{region '#Template'}
	{attribute 'Version' := '1.2.1.0'}
	{attribute 'Tags' := '"LCID": "1031", "Text": "General, Cabinet, Control cabinet, Acknowledgement"'}
	{attribute 'Tags' := '"LCID": "1033", "Text": "General, Cabinet, Control cabinet, Acknowledgement"'}
	{attribute 'Using' := '"Type": "Template", "URI": "EC_AMEV"'}
	{attribute 'Description' := '"LCID": "1031", "Text": "Schaltschrank Quittierung"'}
	{attribute 'Description' := '"LCID": "1033", "Text": "Control cabinet acknowledgement"'}
{endregion}
FUNCTION_BLOCK FB_BA_ControlCabinetBasic EXTENDS FB_BA_View
VAR
	// By default, the entire project structure can be acknowledged.
	// There may be constellations (e.g. multiple control cabinets) where only one part of the project structure (e.g. multiple buildings) has to be acknowledged.
	// > In this case separete parts can be assigned here: 
	iAckView1				: I_BA_View;
	iAckView2				: I_BA_View;
	iAckView3				: I_BA_View;
END_VAR
VAR_INPUT CONSTANT
	LampFault				: FB_BA_ActuatorCmd;		
	AckButton				: FB_BA_CombinationBI_BV;													
	RstHw					: FB_BA_ActuatorCmd;														
END_VAR
VAR				
	bIsDisturbed			: BOOL;
	bHasUnackEvent			: BOOL;
	bBlink					: BOOL;
	tAlmLampImpuls			: FB_BA_Blink;						
	tpResetHw				: TP;	
	rtrigRstSwi				: R_TRIG;
	bTrigRstSwi				: BOOL;
	rtrigRstButton			: R_TRIG;
	bTrigRstButton			: BOOL;	
END_VAR

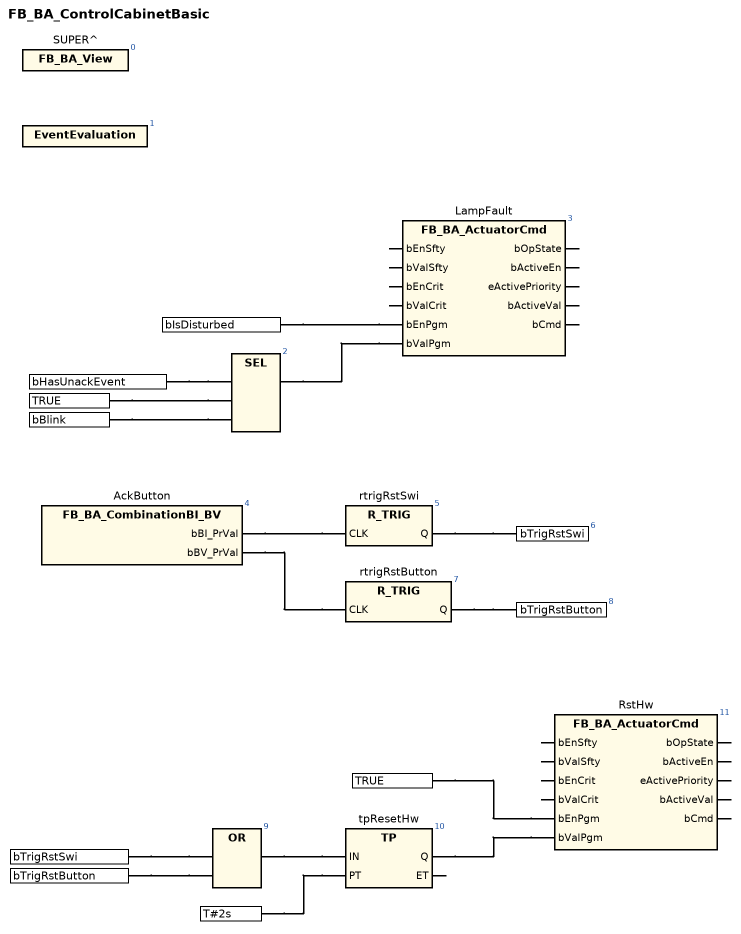
SUPER^(); // FB_BA_View
EventEvaluation();
LampFault(bEnPgm := bIsDisturbed, bValPgm := SEL(bHasUnackEvent, TRUE, bBlink)); // FB_BA_ActuatorCmd
AckButton(); // FB_BA_CombinationBI_BV
rtrigRstSwi(CLK := AckButton.bBI_PrVal); // R_TRIG
bTrigRstSwi := rtrigRstSwi.Q;
rtrigRstButton(CLK := AckButton.bBV_PrVal); // R_TRIG
bTrigRstButton := rtrigRstButton.Q;
tpResetHw(IN := bTrigRstSwi OR bTrigRstButton, PT := T#2s); // TP
RstHw(bEnPgm := TRUE, bValPgm := tpResetHw.Q); // FB_BA_ActuatorCmd

METHOD PRIVATE Ack
VAR_INPUT
	iView			: I_BA_View;
END_VAR
IF (iView <> 0) THEN
	iView.AcknowledgeObjectsPLC := (bTrigRstSwi) OR (bTrigRstButton);	
END_IF
END_METHOD

METHOD PRIVATE EventEvaluation
VAR
	_iView			: I_BA_View;
END_VAR
bIsDisturbed := FALSE;
bHasUnackEvent := FALSE;

IF (iAckView1 = 0) AND (iAckView2 = 0) AND (iAckView3 = 0) THEN
	// Treat project structure via root-object:
	Ack(BA_Globals.Top);
	GetErrors(BA_Globals.Top);
ELSE
	// Treat each defined object:
	Ack(iAckView1);
	GetErrors(iAckView1);
	
	Ack(iAckView2);
	GetErrors(iAckView2);
	
	Ack(iAckView3);
	GetErrors(iAckView3);
END_IF

// Generate alarm lamp impulse:
tAlmLampImpuls();

bBlink := tAlmLampImpuls.bQ;
END_METHOD

METHOD FB_init : BOOL
VAR_INPUT
	bInitRetains : BOOL; // if TRUE, the retain variables are initialized (warm start / cold start)
	bInCopyCode : BOOL;  // if TRUE, the instance afterwards gets moved into the copy code (online change)
END_VAR
LampFault.iParent							:= THIS^;
LampFault.iLabel							:= LblCmpGeneral.ControlCabinet_LampFault;			
LampFault.sObjectName						:= '{Idx=01}';
LampFault.eDPADMode							:= E_BA_DPADMode.eInclude;																						
LampFault.Cmd.iLabel						:= LblCmpGeneral.ControlCabinet_LampFault_Cmd;			
LampFault.Cmd.sObjectName					:= '{Idx=01}';	
LampFault.Cmd.ePolarity						:= E_BA_Polarity.eNormal;
LampFault.Cmd.eFeedbackPolarity				:= E_BA_Polarity.eNormal;
LampFault.Cmd.eOverriddenPolarity			:= E_BA_Polarity.eReverse;
LampFault.Cmd.sActiveText 					:= txtEvent_On;
LampFault.Cmd.sInactiveText 				:= txtEvent_Off;
LampFault.Cmd.nEventClassID					:= EC_ID.NC40;
LampFault.Cmd.aEventTransitionText[1]		:= txtEvent_Disturb;
LampFault.Cmd.aEventTransitionText[2]		:= txtEvent_None;
LampFault.Cmd.aEventTransitionText[3]		:= txtEvent_Normal;
LampFault.Cmd.bEventDetectionEnable			:= FALSE;
LampFault.Cmd.eEnPlantLock					:= E_BA_LockPriority.eNoLock;	

AckButton.iParent							:= THIS^;		
AckButton.iLabel 							:= LblCmpGeneral.ControlCabinet_AckButton;	
AckButton.sObjectName						:= '{Idx=01}';
AckButton.eDPADMode							:= E_BA_DPADMode.eInclude;																						
AckButton.Input.iLabel						:= LblCmpGeneral.ControlCabinet_AckButton_Input;
AckButton.Input.ePolarity					:= E_BA_Polarity.eNormal;
AckButton.Input.bEventDetectionEnable		:= FALSE;
AckButton.Value.iLabel						:= LblCmpGeneral.ControlCabinet_AckButton_Value;
AckButton.Value.eToggleMode 				:= E_BA_ToggleMode.ePushButton;									

RstHw.iParent								:= THIS^;
RstHw.iLabel								:= LblCmpGeneral.ControlCabinet_RstHw;			
RstHw.sObjectName							:= '{Idx=02}';
RstHw.eDPADMode								:= E_BA_DPADMode.eInclude;																						
RstHw.Cmd.iLabel							:= LblCmpGeneral.ControlCabinet_RstHw_Cmd;			
RstHw.Cmd.sObjectName						:= '{Idx=01}';	
RstHw.Cmd.ePolarity							:= E_BA_Polarity.eNormal;
RstHw.Cmd.eFeedbackPolarity					:= E_BA_Polarity.eNormal;
RstHw.Cmd.eOverriddenPolarity				:= E_BA_Polarity.eReverse;
RstHw.Cmd.sActiveText 						:= txtEvent_On;
RstHw.Cmd.sInactiveText 					:= txtEvent_Off;
RstHw.Cmd.nEventClassID						:= EC_ID.NC40;
RstHw.Cmd.aEventTransitionText[1]			:= txtEvent_Disturb;
RstHw.Cmd.aEventTransitionText[2]			:= txtEvent_None;
RstHw.Cmd.aEventTransitionText[3]			:= txtEvent_Normal;
RstHw.Cmd.bEventDetectionEnable				:= FALSE;
RstHw.Cmd.eEnPlantLock						:= E_BA_LockPriority.eNoLock;	

tAlmLampImpuls.bEn							:=	TRUE; 
tAlmLampImpuls.nTiOn						:=	800;
tAlmLampImpuls.nTiOff						:=	800;
END_METHOD

METHOD PRIVATE GetErrors
VAR_INPUT
	iView			: I_BA_View;
END_VAR
VAR
	iTemp			: INT;
	fbEvents		: REFERENCE TO FB_BA_EventIndicator;
END_VAR
IF (iView <> 0) THEN
	fbEvents REF= iView.ActiveEvents;
	
	FOR iTemp := E_BA_EventType.First TO E_BA_EventType.Last DO
		IF (fbEvents.aEventsPerIconImage[iTemp].nCount > 0) THEN
			bIsDisturbed := TRUE;
			
			CASE (fbEvents.aEventsPerIconImage[iTemp].eMostPriorisedState) OF
				E_BA_EventIconState.ePresent,
				E_BA_EventIconState.eGone:
					bHasUnackEvent := TRUE;
			END_CASE
		END_IF
	END_FOR
END_IF
END_METHOD

METHOD PROTECTED Reset
VAR_INPUT
	bUnregister			: BOOL			:= FALSE;
END_VAR
iAckView1 := 0;
iAckView2 := 0;
iAckView3 := 0;

SUPER^.Reset(bUnregister);
END_METHOD

END_FUNCTION_BLOCK

(* stored: Version 1.1.0.1, ProductVersion 3.1.4024.9
   POU FB_BA_ControlCabinetBasic: Id {604963d2-3a97-4043-94de-95d3b4db0240}, SpecialFunc None
   Folder [Private]: Id {3a323497-da88-4433-8f0f-c85eda61d4c2}
   Folder [Protected] Management: Id {ee78fcf5-c643-4757-b0a9-d427f9ffb85f}
   Method Ack: Id {9a3dc274-d6d8-40f3-b953-00a8d78f8fc2}
   Method EventEvaluation: Id {c70da550-f453-4d8a-a859-47362e714857}
   Method FB_init: Id {61127a31-571a-454d-b17b-f86e862d8456}
   Method GetErrors: Id {5b168de7-bf2c-4a2e-88bc-5dd9fb1e29ea}
   Method Reset: Id {b1e7e7cc-326e-425e-b8f2-73072c84f153} *)
